FUNCTION FUN_GetDateWithoutSeperator : STRING
VAR_INPUT
	stNtTime		:TIMESTRUCT;
END_VAR
VAR
	sDate			:STRING;
END_VAR

// Initialize string
sDate := '';

// Add year to string
sDate := UINT_TO_STRING(stNtTime.wYear);

// Add month to string
IF stNtTime.wMonth < 10 THEN
	sDate := CONCAT(sDate,'0');
END_IF
sDate := CONCAT(sDate,UINT_TO_STRING(stNtTime.wMonth));

// Add day to string
IF stNtTime.wDay < 10 THEN
	sDate := CONCAT(sDate, '0');
END_IF
sDate := CONCAT(sDate,UINT_TO_STRING(stNtTime.wDay));

// Return result
FUN_GetDateWithoutSeperator := sDate;

END_FUNCTION

(* stored: Version 1.1.0.1, ProductVersion 3.1.4024.12
   POU FUN_GetDateWithoutSeperator: Id {73d3b13c-8d95-4475-b4fc-81ea9ff6c2c7}, SpecialFunc None *)
